FUNCTION_BLOCK LinTransfo
VAR_INPUT
	fIN				: REAL;
	fIN_min 		: REAL;
	fIN_max			: REAL;
	fOUT_min		: REAL;
	fOUT_max 		: REAL;
END_VAR
VAR_OUTPUT
	fOUT 			: REAL;	
END_VAR
VAR
END_VAR

fOUT := fOUT_min + (fIN - fIN_MIN) * (fOUT_max - fOUT_min) / (fIN_max - fIN_min);

END_FUNCTION_BLOCK

(* stored: Version 1.1.0.1
   POU LinTransfo: Id {f6f13783-b748-42a3-ba0a-5db72e3925f9}, SpecialFunc None *)
